// TwinCAT 3 PLC project Monolitico_PLC
// ProgramVersion: 3.1.4024.0
// libraries:
//   Tc2_Standard, * (Beckhoff Automation GmbH)
//   Tc2_System, * (Beckhoff Automation GmbH)
//   Tc3_Module, * (Beckhoff Automation GmbH)
//   VisuDialogs, * (System)
// project tree:
//   / GlobalTextList.TcGTLO, PlcTask.TcTTO, Visualization Manager.TcVMO (not stored)
//   POUs/ FB_Estacion.TcPOU, MAIN.TcPOU
//   VISUs/ V_Estacion.TcVIS
// real-time tasks:
//   TASK PlcTask: cycle T#10ms, priority 20, ADS port 350
// I/O:
//   DEVICE Device 1 (EtherCAT) (disabled), AmsNetId 192.168.56.1.2.1
//     Term 1 (EK1200) [EK1200-5000 EtherCAT Power supply (2A E-Bus)]
//       Term 1 (EL6910) [EL6910, TwinSAFE PLC]
//       Term 2 (EL1918) [EL1918, 8Ch. Safety Input 24V, TwinSAFE]
//         modules: Module 1 (FSOE), Module 2 (FSLOGIC)
//       Term 3 (EL2904) [EL2904, 4 Ch. Safety Output 24V, 0.5A, TwinSAFE]
//         modules: Module 1 (FSOES), Module 2 (DO)
//       Term 4 (EL1008) [EL1008 8Ch. Dig. Input 24V, 3ms]
//       Term 5 (EL1008) [EL1008 8Ch. Dig. Input 24V, 3ms]
//       Term 6 (EL2008) [EL2008 8Ch. Dig. Output 24V, 0.5A]
//       Term 7 (EL2008) [EL2008 8Ch. Dig. Output 24V, 0.5A]
//       Term 8 (EL1008) [EL1008 8Ch. Dig. Input 24V, 3ms]
//       Term 9 (EL1008) [EL1008 8Ch. Dig. Input 24V, 3ms]
//       Term 10 (EL2008) [EL2008 8Ch. Dig. Output 24V, 0.5A]
//       Term 11 (EL2008) [EL2008 8Ch. Dig. Output 24V, 0.5A]
//       Term 12 (EL9011) [EL9011 End Terminal]
//   DEVICE Device 3 (RT-Ethernet Protocol) (disabled), AmsNetId 192.168.56.1.4.1
//   DEVICE Device 2 (NOV-DP-RAM) (disabled)
// variable links:
//   Monolitico_PLC/Monolitico_PLC Instance <-> Device 1 (EtherCAT)/Term 1 (EK1200)/Term 10 (EL2008)
//     PlcTask Outputs/MAIN.Estacion.o_DescargadorAvanza <-> Channel 1/DescargadorAvanza
//     PlcTask Outputs/MAIN.Estacion.o_DescargadorBaja <-> Channel 3/DescargadorBaja
//     PlcTask Outputs/MAIN.Estacion.o_DescargadorRetrocede <-> Channel 2/DescargadorRetrocede
//     PlcTask Outputs/MAIN.Estacion.o_DescargadorSucciona <-> Channel 8/DescargadorSucciona
//     PlcTask Outputs/MAIN.Estacion.o_DesplazadorAvanza <-> Channel 6/DesplazadorAvanza
//     PlcTask Outputs/MAIN.Estacion.o_EmpujadorAvanza <-> Channel 7/EmpujadorAvanza
//     PlcTask Outputs/MAIN.Estacion.o_RechazadorAvanza <-> Channel 4/RechazadorAvanza
//     PlcTask Outputs/MAIN.Estacion.o_VerificardorBaja <-> Channel 5/VerificadorBaja
//   Monolitico_PLC/Monolitico_PLC Instance <-> Device 1 (EtherCAT)/Term 1 (EK1200)/Term 4 (EL1008)
//     PlcTask Inputs/MAIN.Estacion.i_CodigoPaleBit0 <-> Channel 7/CodigoPaleBit0
//     PlcTask Inputs/MAIN.Estacion.i_CodigoPaleBit1 <-> Channel 8/CodigoPaleBit1
//     PlcTask Inputs/MAIN.Estacion.i_EstacionConectada <-> Channel 5/EstacionConectada
//     PlcTask Inputs/MAIN.Estacion.i_PresenciaPale <-> Channel 6/PresenciaPale
//     PlcTask Inputs/MAIN.Estacion.i_PulsadorEmergencia <-> Channel 1/PulsadorEmergencia
//     PlcTask Inputs/MAIN.Estacion.i_PulsadorMarcha <-> Channel 3/PulsadorMarcha
//     PlcTask Inputs/MAIN.Estacion.i_PulsadorParada <-> Channel 4/PulsadorParada
//     PlcTask Inputs/MAIN.Estacion.i_SelectorManual <-> Channel 2/SelectorManual
//   Monolitico_PLC/Monolitico_PLC Instance <-> Device 1 (EtherCAT)/Term 1 (EK1200)/Term 5 (EL1008)
//     PlcTask Inputs/MAIN.Estacion.i_CodigoPaleBit2 <-> Channel 1/CodigoPaleBit2
//     PlcTask Inputs/MAIN.Estacion.i_DetectorPresion <-> Channel 2/DetectorPresion
//   Monolitico_PLC/Monolitico_PLC Instance <-> Device 1 (EtherCAT)/Term 1 (EK1200)/Term 6 (EL2008)
//     PlcTask Outputs/MAIN.Estacion.o_CintaActiva <-> Channel 5/CintaActiva
//     PlcTask Outputs/MAIN.Estacion.o_CintaInvierte <-> Channel 6/CintaInvierte
//     PlcTask Outputs/MAIN.Estacion.o_DesconectaEstacion <-> Channel 1/DesconectaEstacion
//     PlcTask Outputs/MAIN.Estacion.o_LamparaAlarma <-> Channel 2/LamparaAlarma
//     PlcTask Outputs/MAIN.Estacion.o_LamparaMarcha <-> Channel 3/LamparaMarcha
//     PlcTask Outputs/MAIN.Estacion.o_LamparaMaterial <-> Channel 4/LamparaMaterial
//     PlcTask Outputs/MAIN.Estacion.o_RetenedorBaja <-> Channel 7/RetenedorBaja
//     PlcTask Outputs/MAIN.Estacion.o_SeparadorSube <-> Channel 8/SeparadorSube
//   Monolitico_PLC/Monolitico_PLC Instance <-> Device 1 (EtherCAT)/Term 1 (EK1200)/Term 7 (EL2008)
//     PlcTask Outputs/MAIN.Estacion.o_AvisadorSonoro <-> Channel 1/AvisadorSonoro
//   Monolitico_PLC/Monolitico_PLC Instance <-> Device 1 (EtherCAT)/Term 1 (EK1200)/Term 8 (EL1008)
//     PlcTask Inputs/MAIN.Estacion.i_DescargadorAbajo <-> Channel 4/DescargadorAbajo
//     PlcTask Inputs/MAIN.Estacion.i_DescargadorArriba <-> Channel 3/DescargadorArriba
//     PlcTask Inputs/MAIN.Estacion.i_DescargadorDelante <-> Channel 2/DescargadorDelante
//     PlcTask Inputs/MAIN.Estacion.i_DescargadorDetras <-> Channel 1/DescargadorDetras
//     PlcTask Inputs/MAIN.Estacion.i_DesplazadorDetras <-> Channel 7/DesplazadorDetras
//     PlcTask Inputs/MAIN.Estacion.i_EmpujadorDetras <-> Channel 8/EmpujadorDetras
//     PlcTask Inputs/MAIN.Estacion.i_VerificadorAbajo <-> Channel 6/VerificadorAbajo
//     PlcTask Inputs/MAIN.Estacion.i_VerificadorArriba <-> Channel 5/VerificadorArriba
//   Monolitico_PLC/Monolitico_PLC Instance <-> Device 1 (EtherCAT)/Term 1 (EK1200)/Term 9 (EL1008)
//     PlcTask Inputs/MAIN.Estacion.i_DescargadorVacio <-> Channel 2/DescargadorVacio
//     PlcTask Inputs/MAIN.Estacion.i_EmpujadorDelante <-> Channel 1/EmpujadorDelante
//     PlcTask Inputs/MAIN.Estacion.i_PresenciaBase <-> Channel 3/PresenciaBase

CONFIGURATION Monolitico_PLC
    RESOURCE PLC ON TwinCAT3
        TASK PlcTask(INTERVAL := T#10ms, PRIORITY := 20);
        PROGRAM MAIN WITH PlcTask : MAIN;
    END_RESOURCE
END_CONFIGURATION

// ---- POUs/MAIN.TcPOU
PROGRAM MAIN
VAR
    Estacion: FB_Estacion;
END_VAR

IF NOT Estacion.i_SelectorManual THEN
	Estacion();
END_IF;

END_PROGRAM

// ---- POUs/FB_Estacion.TcPOU
FUNCTION_BLOCK FB_Estacion
VAR_INPUT
    UnidadesSolicitadas: UINT := 1;
    
	TiempoRetenedor: TIME := T#1S;
	TiempoSeparador: TIME := T#1S;
	TiempoEntradaPale: TIME := T#1S;
    TiempoSalidaPale: TIME := T#1S;
    TiempoTransferenciPale: TIME := T#1S;
    
	TiempoVerificacion: TIME := T#1S;
	TiempoDesplazador: TIME := T#2S;
    TiempoRechazador: TIME := T#1S;
END_VAR
VAR_OUTPUT
    CondicionInicial: BOOL;
    MarchaAutorizada: BOOL;
    UnidadesPendientes: UINT;
    
	i_SelectorManual AT %I*: BOOL;
END_VAR
VAR
    DemandaProduccion: BOOL;
    TareaFinalizada: BOOL;
    
    UnidadCorrecta: BOOL;
    
    // Variables de entrada
    i_PulsadorEmergencia AT %I*: BOOL;
    // i_SelectorManual AT %I*: BOOL;
    i_PulsadorMarcha AT %I*: BOOL;
    i_PulsadorParada AT %I*: BOOL := TRUE; // Normalmente cerrado
    i_EstacionConectada AT %I*: BOOL := TRUE;
    i_PresenciaPale AT %I*: BOOL;
    i_CodigoPaleBit0 AT %I*: BOOL;
    i_CodigoPaleBit1 AT %I*: BOOL;
    
    i_CodigoPaleBit2 AT %I*: BOOL;
    i_DetectorPresion AT %I*: BOOL := TRUE;
    
    i_DescargadorDetras AT %I*: BOOL := TRUE;
    i_DescargadorDelante AT %I*: BOOL;
    i_DescargadorArriba AT %I*: BOOL := TRUE;
    i_DescargadorAbajo AT %I*: BOOL;
    i_VerificadorArriba AT %I*: BOOL := TRUE;
    i_VerificadorAbajo AT %I*: BOOL;
    i_DesplazadorDetras AT %I*: BOOL := TRUE;
    i_AlimentadorDetras AT %I*: BOOL := TRUE;
    
    i_AlimentadorDelante AT %I*: BOOL;
    i_DescargadorVacio AT %I*: BOOL;
    i_PresenciaBase AT %I*: BOOL;
    
    // Variables de salida
    o_DesconectaEstacion AT %Q*: BOOL;
    o_LamparaAlarma AT %Q*: BOOL;
    o_LamparaMarcha AT %Q*: BOOL;
    o_LamparaMaterial AT %Q*: BOOL;
    o_CintaActiva AT %Q*: BOOL;
    o_CintaInvierte AT %Q*: BOOL;
    o_RetenedorBaja AT %Q*: BOOL;
    o_SeparadorSube AT %Q*: BOOL;
    
    o_AvisadorSonoro AT %Q*: BOOL;
    
    o_DescargadorAvanza AT %Q*: BOOL;
    o_DescargadorRetrocede AT %Q*: BOOL;
    o_DescargadorBaja AT %Q*: BOOL;
    o_RechazadorAvanza AT %Q*: BOOL;
    o_VerificardorBaja AT %Q*: BOOL;
    o_DesplazadorAvanza AT %Q*: BOOL;
    o_AlimentadorAvanza AT %Q*: BOOL;
    o_DescargadorSucciona AT %Q*: BOOL;
END_VAR

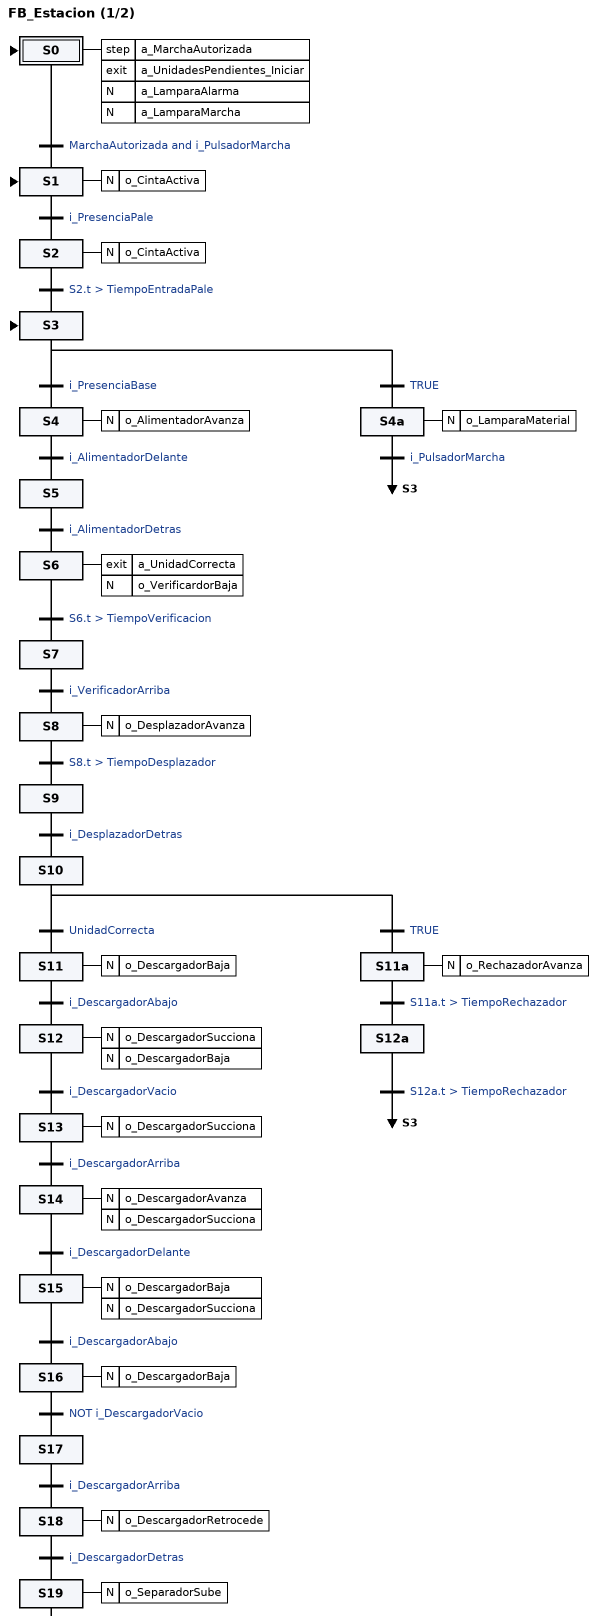
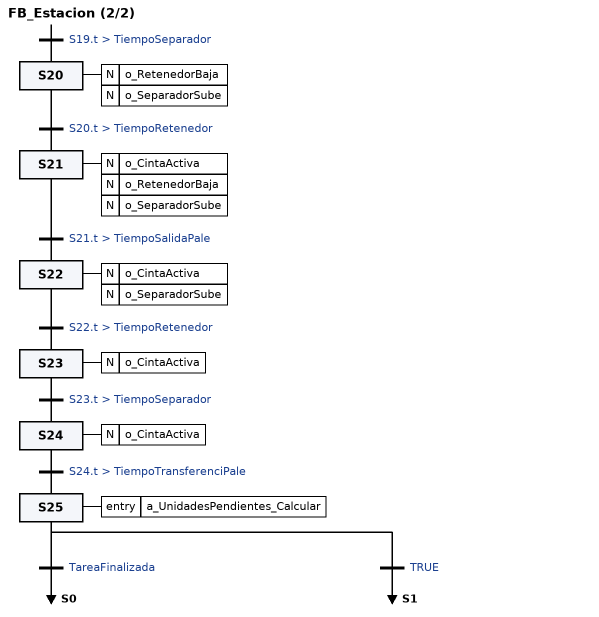
INITIAL_STEP S0:
    a_MarchaAutorizada(N);  // step action
    a_UnidadesPendientes_Iniciar(P0);  // exit action
    a_LamparaAlarma(N);
    a_LamparaMarcha(N);
END_STEP
TRANSITION FROM S0 TO S1
    := MarchaAutorizada and i_PulsadorMarcha;
END_TRANSITION
STEP S1:
    o_CintaActiva(N);
END_STEP
TRANSITION FROM S1 TO S2
    := i_PresenciaPale;
END_TRANSITION
STEP S2:
    o_CintaActiva(N);
END_STEP
TRANSITION FROM S2 TO S3
    := S2.t > TiempoEntradaPale;
END_TRANSITION
STEP S3:
END_STEP
TRANSITION FROM S3 TO S4
    := i_PresenciaBase;
END_TRANSITION
STEP S4:
    o_AlimentadorAvanza(N);
END_STEP
TRANSITION FROM S4 TO S5
    := i_AlimentadorDelante;
END_TRANSITION
STEP S5:
END_STEP
TRANSITION FROM S5 TO S6
    := i_AlimentadorDetras;
END_TRANSITION
STEP S6:
    a_UnidadCorrecta(P0);  // exit action
    o_VerificardorBaja(N);
END_STEP
TRANSITION FROM S6 TO S7
    := S6.t > TiempoVerificacion;
END_TRANSITION
STEP S7:
END_STEP
TRANSITION FROM S7 TO S8
    := i_VerificadorArriba;
END_TRANSITION
STEP S8:
    o_DesplazadorAvanza(N);
END_STEP
TRANSITION FROM S8 TO S9
    := S8.t > TiempoDesplazador;
END_TRANSITION
STEP S9:
END_STEP
TRANSITION FROM S9 TO S10
    := i_DesplazadorDetras;
END_TRANSITION
STEP S10:
END_STEP
TRANSITION FROM S10 TO S11
    := UnidadCorrecta;
END_TRANSITION
STEP S11:
    o_DescargadorBaja(N);
END_STEP
TRANSITION FROM S11 TO S12
    := i_DescargadorAbajo;
END_TRANSITION
STEP S12:
    o_DescargadorSucciona(N);
    o_DescargadorBaja(N);
END_STEP
TRANSITION FROM S12 TO S13
    := i_DescargadorVacio;
END_TRANSITION
STEP S13:
    o_DescargadorSucciona(N);
END_STEP
TRANSITION FROM S13 TO S14
    := i_DescargadorArriba;
END_TRANSITION
STEP S14:
    o_DescargadorAvanza(N);
    o_DescargadorSucciona(N);
END_STEP
TRANSITION FROM S14 TO S15
    := i_DescargadorDelante;
END_TRANSITION
STEP S15:
    o_DescargadorBaja(N);
    o_DescargadorSucciona(N);
END_STEP
TRANSITION FROM S15 TO S16
    := i_DescargadorAbajo;
END_TRANSITION
STEP S16:
    o_DescargadorBaja(N);
END_STEP
TRANSITION FROM S16 TO S17
    := NOT i_DescargadorVacio;
END_TRANSITION
STEP S17:
END_STEP
TRANSITION FROM S17 TO S18
    := i_DescargadorArriba;
END_TRANSITION
STEP S18:
    o_DescargadorRetrocede(N);
END_STEP
TRANSITION FROM S18 TO S19
    := i_DescargadorDetras;
END_TRANSITION
STEP S19:
    o_SeparadorSube(N);
END_STEP
TRANSITION FROM S19 TO S20
    := S19.t > TiempoSeparador;
END_TRANSITION
STEP S20:
    o_RetenedorBaja(N);
    o_SeparadorSube(N);
END_STEP
TRANSITION FROM S20 TO S21
    := S20.t > TiempoRetenedor;
END_TRANSITION
STEP S21:
    o_CintaActiva(N);
    o_RetenedorBaja(N);
    o_SeparadorSube(N);
END_STEP
TRANSITION FROM S21 TO S22
    := S21.t > TiempoSalidaPale;
END_TRANSITION
STEP S22:
    o_CintaActiva(N);
    o_SeparadorSube(N);
END_STEP
TRANSITION FROM S22 TO S23
    := S22.t > TiempoRetenedor;
END_TRANSITION
STEP S23:
    o_CintaActiva(N);
END_STEP
TRANSITION FROM S23 TO S24
    := S23.t > TiempoSeparador;
END_TRANSITION
STEP S24:
    o_CintaActiva(N);
END_STEP
TRANSITION FROM S24 TO S25
    := S24.t > TiempoTransferenciPale;
END_TRANSITION
TRANSITION FROM S10 TO S11a
    := TRUE;
END_TRANSITION
STEP S11a:
    o_RechazadorAvanza(N);
END_STEP
TRANSITION FROM S11a TO S12a
    := S11a.t > TiempoRechazador;
END_TRANSITION
STEP S12a:
END_STEP
TRANSITION FROM S12a TO S3
    := S12a.t > TiempoRechazador;
END_TRANSITION
TRANSITION FROM S3 TO S4a
    := TRUE;
END_TRANSITION
STEP S4a:
    o_LamparaMaterial(N);
END_STEP
TRANSITION FROM S4a TO S3
    := i_PulsadorMarcha;
END_TRANSITION
STEP S25:
    a_UnidadesPendientes_Calcular(P1);  // entry action
END_STEP
TRANSITION FROM S25 TO S0
    := TareaFinalizada;
END_TRANSITION
TRANSITION FROM S25 TO S1
    := TRUE;
END_TRANSITION

ACTION a_CondicionInicial:
CondicionInicial := i_DetectorPresion
    AND i_EstacionConectada
    AND i_AlimentadorDetras
    AND i_VerificadorArriba
    AND i_DesplazadorDetras
    AND i_DescargadorDetras
    AND i_DescargadorArriba;
END_ACTION

ACTION a_LamparaAlarma:
o_LamparaAlarma := (S0.x AND NOT MarchaAutorizada);
END_ACTION

ACTION a_LamparaMarcha:
o_LamparaMarcha := NOT S0.x;
END_ACTION

ACTION a_MarchaAutorizada:
a_CondicionInicial();

DemandaProduccion := (UnidadesSolicitadas > 0);
MarchaAutorizada := CondicionInicial AND DemandaProduccion;
END_ACTION

ACTION a_UnidadCorrecta:
UnidadCorrecta := i_VerificadorAbajo;
END_ACTION

ACTION a_UnidadesPendientes_Calcular:
IF UnidadesPendientes > 0 THEN
    UnidadesPendientes := UnidadesPendientes - 1;
END_IF;

TareaFinalizada := (UnidadesPendientes = 0);
END_ACTION

ACTION a_UnidadesPendientes_Iniciar:
UnidadesPendientes := UnidadesSolicitadas;
END_ACTION

END_FUNCTION_BLOCK

// ---- GlobalTextList.TcGTLO
TEXTLIST GlobalTextList
  843 = '%d'
  6 = '0'
  889 = '1'
  795 = '2'
  434 = 'Abajo'
  387 = 'Activa'
  885 = 'Alarma'
  83 = 'Arriba'
  897 = 'Avanza'
  952 = 'Avisador'
  738 = 'Baja'
  35 = 'CI'
  221 = 'Cinta'
  118 = 'Conectada'
  522 = 'Código'
  1 = 'Delante'
  271 = 'Descargador'
  378 = 'Desconecta'
  868 = 'Desplazador'
  232 = 'Detras'
  740 = 'Emergencia'
  90 = 'Empujador'
  111 = 'Entradas y '
  270 = 'Entradas y Salidas'
  578 = 'FMS-201'
  770 = 'inta'
  402 = 'Invierte'
  329 = 'Manual'
  847 = 'Marcha'
  215 = 'Material'
  388 = 'Monolítico'
  601 = 'Palé'
  665 = 'Panel Operador'
  763 = 'Parada'
  560 = 'Pendientes'
  425 = 'Pieza Correcta'
  170 = 'Preseancia'
  173 = 'Presencia'
  974 = 'Presión'
  33 = 'Rechazador'
  269 = 'Retenedor'
  53 = 'Retrocede'
  322 = 'Separador'
  129 = 'Solicitadas'
  529 = 'Sube'
  42 = 'Succiona'
  282 = 'Tarea'
  628 = 'Vacío'
  874 = 'Verificador'
END_TEXTLIST

// ---- VISUs/V_Estacion.TcVIS
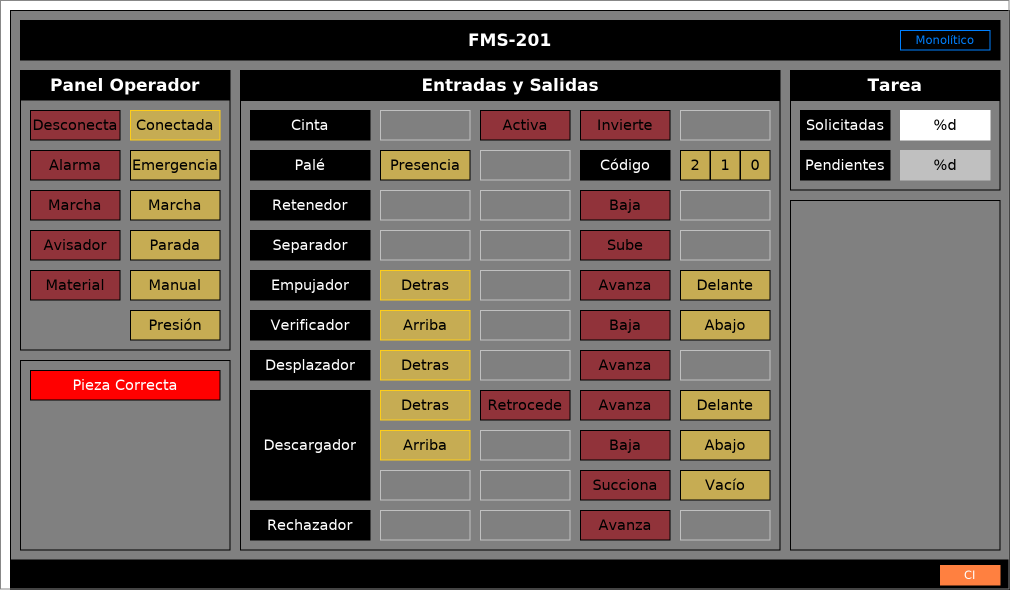
VISUALIZATION V_Estacion  // 1010x590
    Rectangle (10,10 1000x550)
    Rectangle (240,100 540x450)
    Rectangle (20,70 210x280)
    Rectangle (30,110 90x30), "Desconecta"
        tap MAIN.Estacion.o_DesconectaEstacion
    Rectangle (30,150 90x30), "Alarma"
        toggle MAIN.Estacion.o_LamparaAlarma
    Rectangle (30,190 90x30), "Marcha"
        toggle MAIN.Estacion.o_LamparaMarcha
    Rectangle (30,230 90x30), "Avisador"
        tap MAIN.Estacion.o_AvisadorSonoro
    Rectangle (30,270 90x30), "Material"
        toggle MAIN.Estacion.o_LamparaMaterial
    Rectangle (130,110 90x30), "Conectada"
        toggle MAIN.Estacion.i_EstacionConectada
    Rectangle (130,150 90x30), "Emergencia"
        toggle MAIN.Estacion.i_PulsadorEmergencia
    Rectangle (130,190 90x30), "Marcha"
        tap MAIN.Estacion.i_PulsadorMarcha
    Rectangle (130,230 90x30), "Parada"
        tap MAIN.Estacion.i_PulsadorParada p1329445385=TRUE
    Rectangle (130,270 90x30), "Manual"
        toggle MAIN.Estacion.i_SelectorManual
    Rectangle (20,70 210x30), "Panel Operador"
    Rectangle (240,70 540x30), "Entradas y Salidas"
    Rectangle (250,110 120x30), "Cinta"
    Rectangle (250,150 120x30), "Palé"
    Rectangle (250,190 120x30), "Retenedor"
    Rectangle (250,230 120x30), "Separador"
    Rectangle (250,390 120x110), "Descargador"
    Rectangle (250,510 120x30), "Rechazador"
    Rectangle (250,310 120x30), "Verificador"
    Rectangle (250,350 120x30), "Desplazador"
    Rectangle (250,270 120x30), "Empujador"
    Rectangle (480,110 90x30), "Activa"
        toggle MAIN.Estacion.o_CintaActiva
    Rectangle (380,110 90x30)
    Rectangle (580,110 90x30), "Invierte"
        toggle MAIN.Estacion.o_CintaInvierte
    Rectangle (680,110 90x30)
    Rectangle (380,150 90x30), "Presencia"
        toggle MAIN.Estacion.i_PresenciaPale
    Rectangle (480,150 90x30)
    Rectangle (580,150 90x30), "Código"
    Rectangle (680,150 30x30), "2"
        toggle MAIN.Estacion.i_CodigoPaleBit2
    Rectangle (710,150 30x30), "1"
        toggle MAIN.Estacion.i_CodigoPaleBit1
    Rectangle (740,150 30x30), "0"
        toggle MAIN.Estacion.i_CodigoPaleBit0
    Rectangle (380,190 90x30)
    Rectangle (580,190 90x30), "Baja"
        toggle MAIN.Estacion.o_RetenedorBaja
    Rectangle (680,190 90x30)
    Rectangle (480,230 90x30)
    Rectangle (580,230 90x30), "Sube"
        toggle MAIN.Estacion.o_SeparadorSube
    Rectangle (380,230 90x30)
    Rectangle (680,230 90x30)
    Rectangle (580,270 90x30), "Avanza"
        toggle MAIN.Estacion.o_EmpujadorAvanza
    Rectangle (380,270 90x30), "Detras"
        toggle MAIN.Estacion.i_EmpujadorDetras
    Rectangle (480,270 90x30)
    Rectangle (580,310 90x30), "Baja"
        toggle MAIN.Estacion.o_VerificardorBaja
    Rectangle (480,310 90x30)
    Rectangle (580,350 90x30), "Avanza"
        toggle MAIN.Estacion.o_DesplazadorAvanza
    Rectangle (580,390 90x30), "Avanza"
        toggle MAIN.Estacion.o_DescargadorAvanza
    Rectangle (480,390 90x30), "Retrocede"
        toggle MAIN.Estacion.o_DescargadorRetrocede
    Rectangle (480,190 90x30)
    Rectangle (580,430 90x30), "Baja"
        toggle MAIN.Estacion.o_DescargadorBaja
    Rectangle (580,470 90x30), "Succiona"
        toggle MAIN.Estacion.o_DescargadorSucciona
    Rectangle (580,510 90x30), "Avanza"
        toggle MAIN.Estacion.o_RechazadorAvanza
    Rectangle (480,510 90x30)
    Rectangle (480,350 90x30)
    Rectangle (480,430 90x30)
    Rectangle (480,470 90x30)
    Rectangle (680,270 90x30), "Delante"
        toggle MAIN.Estacion.i_EmpujadorDelante
    Rectangle (380,310 90x30), "Arriba"
        toggle MAIN.Estacion.i_VerificadorArriba
    Rectangle (680,310 90x30), "Abajo"
        toggle MAIN.Estacion.i_VerificadorAbajo
    Rectangle (380,350 90x30), "Detras"
        toggle MAIN.Estacion.i_DesplazadorDetras
    Rectangle (680,350 90x30)
    Rectangle (680,510 90x30)
    Rectangle (380,510 90x30)
    Rectangle (380,470 90x30)
    Rectangle (380,390 90x30), "Detras"
        toggle MAIN.Estacion.i_DescargadorDetras
    Rectangle (680,390 90x30), "Delante"
        toggle MAIN.Estacion.i_DescargadorDelante
    Rectangle (380,430 90x30), "Arriba"
        toggle MAIN.Estacion.i_DescargadorArriba
    Rectangle (680,430 90x30), "Abajo"
        toggle MAIN.Estacion.i_DescargadorAbajo
    Rectangle (680,470 90x30), "Vacío"
        toggle MAIN.Estacion.i_DescargadorVacio
    Rectangle (20,20 980x40), "FMS-201"
    Rectangle (20,360 210x190)
    Rectangle (900,30 90x20), "Monolítico"
    Rectangle (130,310 90x30), "Presión"
        toggle MAIN.Estacion.i_DetectorPresion
    Rectangle (10,560 1000x30)
    Rectangle (940,565 60x20), "CI", colour toggle: MAIN.Estacion.CondicionInicial
    Rectangle (30,370 190x30), "Pieza Correcta", colour toggle: MAIN.Estacion.CondicionInicial
    Rectangle (790,100 210x90)
    Rectangle (790,70 210x30), "Tarea"
    Rectangle (790,200 210x350)
    Rectangle (800,110 90x30), "Solicitadas"
    Rectangle (800,150 90x30), "Pendientes"
    Rectangle (900,110 90x30), "%d", text variable: MAIN.Estacion.ManiobrasSolicitadas
        OnMouseClick: write the text variable via Default
    Rectangle (900,150 90x30), "%d", text variable: MAIN.Estacion.ManiobrasPendientes
END_VISUALIZATION
